Fanuc KAREL source: KT00325.KL

PROGRAM KT00325
%NOLOCKGROUP
VAR
  P1: JOINTPOS
  P2: XYZWPREXT
  OUT: BOOLEAN
BEGIN
    P2.Y = 2.0
  OUT = P1 <> P2
END KT00325
